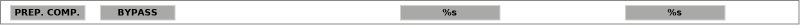
VISUALIZATION Header_2  // 800x25
    Textfield (400,5 75x15), "PREP. COMP."
    Textfield (100,5 75x15), "BYPASS"
    Textfield (400,5 100x15), "%s", text variable: HMI_Global.sSystemDate
    Textfield (625,5 100x15), "%s", text variable: HMI_Global.sSystemTime
    Textfield (10,5 75x15), "PREP. COMP."
END_VISUALIZATION

(* stored: Version 1.1.0.1, ProductVersion 3.1.4024.12
   Visu Header_2: Id {aa1b33aa-45cd-42a5-ab6d-0c8d88f25650} *)
